(* CODESYS project GVL_DETAIL.gvl.xml

Project tree, tasks and I/O mapping:
  global variables GVL_DETAIL
*)

// GVL_DETAIL
{attribute 'qualified_only'}
VAR_GLOBAL
	arrDetail : ARRAY [1..GVL_CELL_SETTINGS.NumberDetail] OF ST_DETAIL; // Содержимое слотов магазина
END_VAR
